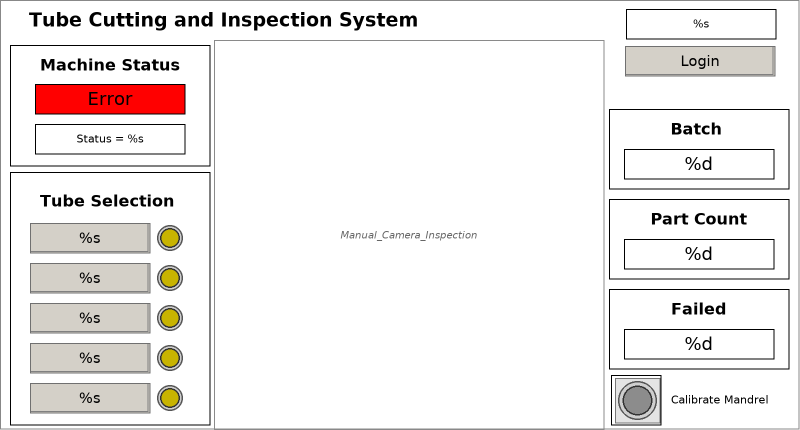
VISUALIZATION Front_Panel  // 800x430
    Rectangle (611,375 50x50), colour toggle: MAIN.fbSlitter.Manual.bCalibrateMandrel
    Frame (214,40 390x390)
        shows Manual_Camera_Inspection()
    Rectangle (10,172 200x253)
    Label (10,186 200x30), "Tube Selection"
    Button (30,223 120x30), "%s", text variable: MAIN.TubeSelection[1].ProductName
        OnMouseClick: execute {
            MAIN.TubeIndicator[1] := TRUE;
            MAIN.TubeIndicator[2] := FALSE;
            MAIN.TubeIndicator[3] := FALSE;
            MAIN.TubeIndicator[4] := FALSE;
            MAIN.TubeIndicator[5] := FALSE;
        }
    Button (30,343 120x30), "%s", text variable: MAIN.TubeSelection[4].ProductName, input disabled if: TRUE
        OnMouseClick: execute {
            MAIN.TubeIndicator[1] := FALSE;
            MAIN.TubeIndicator[2] := FALSE;
            MAIN.TubeIndicator[3] := FALSE;
            MAIN.TubeIndicator[4] := TRUE;
            MAIN.TubeIndicator[5] := FALSE;
        }
    Button (30,383 120x30), "%s", text variable: MAIN.TubeSelection[5].ProductName, input disabled if: TRUE
        OnMouseClick: execute {
            MAIN.TubeIndicator[1] := FALSE;
            MAIN.TubeIndicator[2] := FALSE;
            MAIN.TubeIndicator[3] := FALSE;
            MAIN.TubeIndicator[4] := FALSE;
            MAIN.TubeIndicator[5] := TRUE;
        }
    Lamp1 (155,223 30x30), variable: MAIN.TubeIndicator[1], style: Lamp-Lamp1-Yellow
    Lamp1 (155,263 30x30), variable: MAIN.TubeIndicator[2], style: Lamp-Lamp1-Yellow
    Lamp1 (155,303 30x30), variable: MAIN.TubeIndicator[3], style: Lamp-Lamp1-Yellow
    Lamp1 (155,343 30x30), variable: MAIN.TubeIndicator[4], style: Lamp-Lamp1-Yellow
    Lamp1 (155,383 30x30), variable: MAIN.TubeIndicator[5], style: Lamp-Lamp1-Yellow
    Label (0,5 800x30), "Tube Cutting and Inspection System"
    Rectangle (10,45 200x121)
    Label (10,50 200x30), "Machine Status"
    Rectangle (35,84 150x30), "Initializing", invisible if: MAIN.eState <> E_PMLState.ePMLState_Clearing
    Rectangle (35,84 150x30), "Ready", invisible if: MAIN.eState <> E_PMLState.ePMLState_Idle
    Rectangle (35,84 150x30), "Running", invisible if: MAIN.eState <> E_PMLState.ePMLState_Execute
    Rectangle (35,84 150x30), "Error", invisible if: MAIN.eState <> E_PMLState.ePMLState_Aborted
    Rectangle (609,109 180x80)
    Label (609,114 180x30), "Batch"
    Rectangle (624,149 150x30), "%d", text variable: MAIN.iBatch
        OnMouseClick: write MAIN.hmiBatch via Default, title 'Batch Number'
    Rectangle (609,199 180x80)
    Label (609,204 180x30), "Part Count"
    Rectangle (624,239 150x30), "%d", text variable: MAIN.iCounter
    Rectangle (609,289 180x80)
    Label (609,294 180x30), "Failed"
    Rectangle (624,329 150x30), "%d", text variable: MAIN.iCountFailed
    Rectangle (35,124 150x30), "Status = %s", text variable: MAIN.hmiStatus
    Rectangle (626,9 150x30), "%s", text variable: MAIN.currentUser
    Button (625,46 150x30), "Login"
        OnMouseClick: VisuUserMgmt Type=Login
    PushSwitch (615,378 45x45), variable: MAIN.fbSlitter.Manual.bCalibrateMandrel, behaviour: TOGGLE, style: Switch-PushSwitch-Gray
    Label (668,385 111x30), "Calibrate Mandrel"
    Button (30,263 120x30), "%s", text variable: MAIN.TubeSelection[2].ProductName
        OnMouseClick: execute {
            MAIN.TubeIndicator[1] := FALSE;
            MAIN.TubeIndicator[2] := TRUE;
            MAIN.TubeIndicator[3] := FALSE;
            MAIN.TubeIndicator[4] := FALSE;
            MAIN.TubeIndicator[5] := FALSE;
        }
    Button (30,303 120x30), "%s", text variable: MAIN.TubeSelection[3].ProductName
        OnMouseClick: execute {
            MAIN.TubeIndicator[1] := FALSE;
            MAIN.TubeIndicator[2] := FALSE;
            MAIN.TubeIndicator[3] := TRUE;
            MAIN.TubeIndicator[4] := FALSE;
            MAIN.TubeIndicator[5] := FALSE;
        }
END_VISUALIZATION

(* stored: Version 1.1.0.1, ProductVersion 3.1.4024.9
   Visu Front_Panel: Id {435784a8-d968-4497-b3f7-11a3e0bc9722} *)
